(*
    This is the main program for execution of the unit tests.
*)
PROGRAM PRG_TEST
VAR	
    (* Test function blocks *)
    fbDiagnosticMessageDiagnosticCodeParser_Test : FB_DiagnosticMessageDiagnosticCodeParser_Test;
    fbDiagnosticMessageFlagsParser_Test : FB_DiagnosticMessageFlagsParser_Test;
    fbDiagnosticMessageParser_Test : FB_DiagnosticMessageParser_Test;
    fbDiagnosticMessageTextIdentityParser_Test : FB_DiagnosticMessageTextIdentityParser_Test;
    fbDiagnosticMessageTimeStampParser_Test : FB_DiagnosticMessageTimeStampParser_Test;
END_VAR

TcUnit.RUN();

END_PROGRAM

(* stored: Version 1.1.0.1, ProductVersion 3.1.4022.18
   POU PRG_TEST: Id {0e87b1b9-66e8-4e1a-b53f-6926a5ea0301}, SpecialFunc None *)
